// TwinCAT 3 PLC project Untitled1
// ProgramVersion: 3.1.4026.16
// libraries:
//   Tc2_MC2, * (Beckhoff Automation GmbH)
//   Tc2_Standard, * (Beckhoff Automation GmbH)
//   Tc2_System, * (Beckhoff Automation GmbH)
// project tree:
//   / PlcTask.TcTTO
//   POUs/ f_noteDecoder.TcPOU, MAIN.TcPOU, fb_MUZIK_Parser.TcPOU, nota_hiz_donusturucu.TcPOU, STRING_in_ARRAY.TcPOU
// real-time tasks:
//   TASK PlcTask: cycle T#10ms, priority 20, ADS port 350

CONFIGURATION Untitled1
    RESOURCE PLC ON TwinCAT3
        TASK PlcTask(INTERVAL := T#10ms, PRIORITY := 20);
        PROGRAM MAIN WITH PlcTask : MAIN;
    END_RESOURCE
END_CONFIGURATION

// ---- POUs/MAIN.TcPOU
PROGRAM MAIN
VAR
	b_butonlar 	: ARRAY[1..15] OF BOOL;
	r_zamanlar 	: ARRAY[1..15] OF REAL;
	b_togglelar : ARRAY[1..15] OF BOOL;
	b_scale		: ARRAY[1..12] OF BOOL;

	r_key		: REAL;

	i			: INT;
	j 			: INT := 1;
	k			: INT := 1;
	key_count	: INT;
	last_key	: INT;
	direction   : INT := 1;
	style		: INT;
	b_style		: BOOL;
	b_oldStyle  : BOOL;

	r_mm 		: REAL;
	r_offset	: REAL;
	r_Timer		: REAL;

	mcPower		:MC_Power;
	motor1		:AXIS_REF;
	mcJog		:MC_Jog;
	r_acceleration : REAL := 90000;
	r_deceleration : REAL := 40000;

	b_Manuel  	: BOOL;
	b_vibrato	: BOOL;
	b_Muzik		: BOOL;
	b_Otomatik	: BOOL;
	b_Major		: BOOL := TRUE;

	s_MajorMinor: STRING := 'Major';
	b_ScaleMajor: ARRAY[1..12] OF BOOL := [TRUE, FALSE, TRUE, FALSE, TRUE, TRUE, FALSE, TRUE, FALSE, TRUE, FALSE, TRUE];
	b_ScaleMinor: ARRAY[1..12] OF BOOL := [TRUE, FALSE, TRUE, TRUE, FALSE, TRUE, FALSE, TRUE, TRUE, FALSE, TRUE, FALSE];

	MUZIK_BPS 	: REAL := 10;
	OTOMATIK_BPS: REAL := 1;

	r_BPMTimer 	: REAL;
	r_timerOffset : REAL;
	r_noteTimer	: REAL;

	MUZIK_Parser : fb_MUZIK_Parser;

	MuzikCalmaTuru : BOOL := TRUE;

	(* Offset = -2 yap *)
	MUZIK		: ARRAY[1..100] OF REAL := [1, 1, 1, 5, 5, 5, 8, 8, 6, 6, 6, 10, 10, 10, 13, 13, 1, 1, 1, 5, 5, 5, 8, 8, 6, 13, 12, 13, 12, 13, 8, 5, 1, 1, 1, 5, 5, 5, 8, 8, 6, 6, 6, 10, 10, 10, 13, 13, 1, 1, 16, 16, 16, 15, 15, 15, 13, 13, 13, 8, 7, 8, 7, 4, -1];
	M_TETRIS 	: STRING(255)	 := ['A - E F G - F E D - D F A - G F E - - F G - A - F - D - D -*4 G - Bb D2 - C2 Bb A - - F A - G F E - E F G - A - F - D - D -*3'];
	M_CANAKKALE	: STRING(512) := ['E - Fs*2 -*2 Fs - Fs*10 E2*4 Eb2 E2 Eb2*3 E2*3 Db2*7 D2 Db2 B*3 Db2*6 Eb2*6 E2*6 Db2*6 B*19 -*5 B*3 Db2*3 -*3 Db2*2 - Db2*5 - Db2*3 B*2 - B*5 - B C2*2 B C2 B A*3 Ab*3 A*5 - Ab*3 A*3 B*3 A*3 C2*3 B*3 A*3 Ab*3 Fs*9 E*3 Ab*3 A*3 B*3 Db2*3 -*3 A*5 - Ab*2 - Ab*2 - Fs*8 - Fs*12 - Fs -*18'];
END_VAR

IF NOT (b_Muzik OR b_Otomatik) THEN
	r_mm := 0;
END_IF

(* Piyano tuşlarıyla çalma *)
IF b_Manuel THEN
	FOR i := 1 TO 15 DO
		IF b_butonlar[i] THEN
			r_zamanlar[i] := r_zamanlar[i] + 0.01;
	
			IF i = 1 THEN
				r_mm := nota_hiz_donusturucu(i, r_offset);
			ELSE
				IF (r_zamanlar[i] < r_zamanlar[i-1] AND r_zamanlar[i-1] > 0) OR r_zamanlar[i-1] = 0 THEN
					r_mm := nota_hiz_donusturucu(i, r_offset);
				END_IF
			END_IF
		ELSE
			r_zamanlar[i] := 0;
		END_IF
	END_FOR
END_IF



(* MUZIK'te kayıtlı müziği çalma  -----ESKI----- *)
IF b_Muzik AND NOT MuzikCalmaTuru THEN
	r_BPMTimer := r_BPMTimer + 0.01;
	IF r_BPMTimer > 1/MUZIK_BPS THEN
		r_BPMTimer := 0;
		j := j + 1;
	END_IF

	IF MUZIK[j] = -1 THEN
		j := 1;
	END_IF
	IF MUZIK[j] > 0 THEN
		r_MM := nota_hiz_donusturucu(MUZIK[j], r_offset);
	END_IF
END_IF



(* Daha iyi müzik çalar *)
IF b_Muzik AND MuzikCalmaTuru THEN
	r_offset := -2;
	IF r_noteTimer > 0 THEN
		r_noteTimer := r_noteTimer - 0.01;
	END_IF

	r_BPMTimer := r_BPMTimer + 0.01;
	IF r_BPMTimer > 1/MUZIK_BPS + SEL(r_mm = 0, 0, r_timerOffset) THEN
		r_BPMTimer := SEL(r_mm = 0, 0.0, r_timerOffset);
		MUZIK_Parser(
			MUZIK 		:= M_CANAKKALE,
			i_next 		:= TRUE,
			r_OFFSET	:= r_offset,
			b_stop 		:= FALSE,);
	END_IF
	IF MUZIK_Parser.newNote THEN
		r_noteTimer := 0.02;
	END_IF
	r_MM := MUZIK_Parser.r_mm + ((r_noteTimer) * -6000);
END_IF



(* Anahtar ve gam  *)
r_key := 0;
FOR i := 1 TO 12 DO
	IF b_scale[i] THEN
		r_key := i;
	END_IF
END_FOR

IF r_key > 0 THEN
	FOR i := 0 TO 11 DO
		key_count := REAL_TO_INT(r_key) + i;
		IF key_count > 12 THEN
			key_count := key_count - 12;
		END_IF
		IF b_Major THEN
			b_togglelar[key_count] := b_ScaleMajor[i+1];
		ELSE
			b_togglelar[key_count] := b_ScaleMinor[i+1];
		END_IF
	END_FOR
	b_togglelar[13] := b_togglelar[1];
	b_togglelar[14] := FALSE;
	b_togglelar[15] := FALSE;
END_IF


IF b_style AND NOT b_oldStyle THEN
	IF style > 1 THEN
		style := 0;
	ELSE
		style := style + 1;
	END_IF
END_IF
b_oldStyle := b_style;

(* Otomatik arpej *)
s_MajorMinor := SEL(b_Major, 'Minor', 'Major');
IF b_Otomatik THEN


	IF r_BPMTimer > 1/OTOMATIK_BPS THEN
		r_BPMTimer := 0;

		key_count := 0;
		REPEAT
			k := k + direction;
			IF k > 15 OR k < 1 THEN
				CASE style OF
					0 :
						k := 1;
						direction :=1;
					1 :
						k := 15;
						direction := -1;
					2 :
						direction := -direction;
						k := k + 2*direction;
				END_CASE
			END_IF
			key_count := key_count + 1;
		UNTIL  key_count > 20 OR (b_togglelar[k] AND last_key <> k)
		END_REPEAT
	END_IF
	IF b_togglelar[k] THEN
		last_key := k;
		r_mm := nota_hiz_donusturucu(k, r_offset);
	ELSE
		r_mm := 0;
	END_IF
	r_BPMTimer := r_BPMTimer + 0.01;
END_IF



(* Vibrato *)
IF b_vibrato AND r_mm > 0 THEN
	r_mm := LIMIT(0, r_mm + SIN(r_timer * 360*8 * (pi/180)) * 200, 8800);
END_IF
r_Timer := r_Timer + 0.01;




mcPower(
	Axis:= motor1,
	Enable:= TRUE,
	Enable_Positive:= TRUE,
	Enable_Negative:= TRUE,
	Override:= r_mm/9000 * 100,
	BufferMode:= MC_Aborting);

mcJog(
	Axis:= motor1,
	JogForward:= (r_mm > 0) AND mcPower.Status,
	JogBackwards:= FALSE,
	Mode:= MC_JOGMODE_CONTINOUS,
	Position:= 0,
	Velocity:= 9000,
	Acceleration:= r_acceleration,
	Deceleration:= r_deceleration,
	Jerk:= 900000);

END_PROGRAM

// ---- POUs/fb_MUZIK_Parser.TcPOU
FUNCTION_BLOCK fb_MUZIK_Parser
VAR_INPUT
	MUZIK 		: STRING(512);
	i_next 		: BOOL;
	r_OFFSET	: REAL;
	b_stop   	: BOOL := TRUE;
END_VAR
VAR_OUTPUT
	r_mm 		: REAL;
	newNote		: BOOL;
END_VAR
VAR
	char 		: STRING(4);
	s_reading	: STRING;
	s_NOTE		: STRING;
	r_OCTAVE	: REAL;
	s_OCTARR	: ARRAY[1..10] OF STRING(4) := ['0', '1', '2'];
	i			: INT;
	i_counter	: INT;
END_VAR

IF i_next THEN
	i_counter := i_counter - 1;

	IF i_counter < 1 THEN
		newNote := TRUE;
		s_reading := '';
		r_OCTAVE := 1;
		REPEAT
			i := i + 1;
			char := MID(MUZIK, 1, i);
			IF STRING_in_ARRAY(char, s_OCTARR) THEN
				r_OCTAVE := STRING_TO_REAL(char);
			ELSE
				s_reading := CONCAT(s_reading, char);
			END_IF
		UNTIL MID(MUZIK, 1, i+1) = ' ' OR MID(MUZIK, 1, i+1) = '*' OR i+1 > LEN(MUZIK)
		END_REPEAT

		i := i + 1;

		IF i >= LEN(MUZIK) THEN
			i := 0;
		END_IF

		s_NOTE := s_reading;

		IF MID(MUZIK, 1, i) = '*' THEN
			s_reading := '';
			REPEAT
				i := i + 1;
				char := MID(MUZIK, 1, i);
				s_reading := CONCAT(s_reading, char);
			UNTIL MID(MUZIK, 1, i+1) = ' ' OR i+1 > LEN(MUZIK)
			END_REPEAT
			i := i + 1;
			IF i >= LEN(MUZIK) THEN
				r_mm := 0;
				i:= 0;
			END_IF

			i_counter := STRING_TO_INT(s_reading);
		END_IF
	ELSE
		newNote := FALSE;
	END_IF

	IF s_NOTE = '-' OR s_NOTE = 'x' THEN
		newNote := FALSE;
		IF b_stop THEN
			r_mm := 0;
		END_IF
	ELSE
		r_mm := f_noteDecoder(s_NOTE, r_OCTAVE, r_OFFSET);
	END_IF
END_IF

END_FUNCTION_BLOCK

// ---- POUs/STRING_in_ARRAY.TcPOU
FUNCTION STRING_in_ARRAY : BOOL
VAR_INPUT
	s_STRING 	: STRING;
	s_ARRAY		: ARRAY[1..10] OF STRING(4);
END_VAR
VAR
	i 			: INT;
END_VAR

FOR i := 1 TO 10 DO
	IF s_ARRAY[i] = s_STRING THEN
		STRING_in_ARRAY := TRUE;
		RETURN;
		
	ELSIF s_ARRAY[i] = '' THEN
		STRING_in_ARRAY := FALSE;
		RETURN;
	END_IF
END_FOR

STRING_in_ARRAY := FALSE;
RETURN;

END_FUNCTION

// ---- POUs/f_noteDecoder.TcPOU
FUNCTION f_noteDecoder : REAL
VAR_INPUT
	s_NOTE 		: STRING;
	r_OCTAVE	: REAL;	
	r_OFFSET	: REAL;
END_VAR
VAR
	nota_01 : ARRAY[1..10] OF STRING(4)  := ['0', 'DO', 'C'];
	nota_02 : ARRAY[1..10] OF STRING(4)  := ['1', 'DO#', 'DOd', 'DOs', 'C#', 'Cd', 'Cs', 'REb', 'Db'];
	nota_03 : ARRAY[1..10] OF STRING(4)  := ['2', 'RE', 'D'];
	nota_04 : ARRAY[1..10] OF STRING(4)  := ['3', 'RE#', 'REd', 'REs', 'D#', 'Dd', 'Ds', 'MIb', 'Eb'];
	nota_05 : ARRAY[1..10] OF STRING(4)  := ['4', 'MI', 'E'];
	nota_06 : ARRAY[1..10] OF STRING(4)  := ['5', 'FA', 'F'];
	nota_07 : ARRAY[1..10] OF STRING(4)  := ['6', 'FA#', 'FAd', 'FAs', 'F#', 'Fd', 'Fs', 'SOLb', 'Gb'];
	nota_08 : ARRAY[1..10] OF STRING(4)  := ['7', 'SOL', 'G'];
	nota_09 : ARRAY[1..10] OF STRING(4)  := ['8', 'SOL#', 'SOLd', 'SOLs', 'G#', 'Gd', 'Gs', 'LAb', 'Ab'];
	nota_10 : ARRAY[1..10] OF STRING(4)  := ['9', 'LA', 'A'];
	nota_11 : ARRAY[1..10] OF STRING(4)  := ['10', 'LA#', 'LAd', 'LAs', 'A#', 'Ad', 'As', 'SIb', 'Bb'];
	nota_12 : ARRAY[1..10] OF STRING(4)  := ['11', 'SI', 'B'];
END_VAR

r_OCTAVE := r_OCTAVE - 1;
IF    STRING_in_ARRAY(s_NOTE, nota_01) THEN
	f_noteDecoder := nota_hiz_donusturucu(1  + (12 * r_OCTAVE), r_OFFSET);
ELSIF STRING_in_ARRAY(s_NOTE, nota_02) THEN
	f_noteDecoder := nota_hiz_donusturucu(2  + (12 * r_OCTAVE), r_OFFSET);
ELSIF STRING_in_ARRAY(s_NOTE, nota_03) THEN
	f_noteDecoder := nota_hiz_donusturucu(3  + (12 * r_OCTAVE), r_OFFSET);
ELSIF STRING_in_ARRAY(s_NOTE, nota_04) THEN
	f_noteDecoder := nota_hiz_donusturucu(4  + (12 * r_OCTAVE), r_OFFSET);
ELSIF STRING_in_ARRAY(s_NOTE, nota_05) THEN
	f_noteDecoder := nota_hiz_donusturucu(5  + (12 * r_OCTAVE), r_OFFSET);
ELSIF STRING_in_ARRAY(s_NOTE, nota_06) THEN
	f_noteDecoder := nota_hiz_donusturucu(6  + (12 * r_OCTAVE), r_OFFSET);
ELSIF STRING_in_ARRAY(s_NOTE, nota_07) THEN
	f_noteDecoder := nota_hiz_donusturucu(7  + (12 * r_OCTAVE), r_OFFSET);
ELSIF STRING_in_ARRAY(s_NOTE, nota_08) THEN
	f_noteDecoder := nota_hiz_donusturucu(8  + (12 * r_OCTAVE), r_OFFSET);
ELSIF STRING_in_ARRAY(s_NOTE, nota_09) THEN
	f_noteDecoder := nota_hiz_donusturucu(9  + (12 * r_OCTAVE), r_OFFSET);
ELSIF STRING_in_ARRAY(s_NOTE, nota_10) THEN
	f_noteDecoder := nota_hiz_donusturucu(10 + (12 * r_OCTAVE), r_OFFSET);
ELSIF STRING_in_ARRAY(s_NOTE, nota_11) THEN
	f_noteDecoder := nota_hiz_donusturucu(11 + (12 * r_OCTAVE), r_OFFSET);
ELSIF STRING_in_ARRAY(s_NOTE, nota_12) THEN
	f_noteDecoder := nota_hiz_donusturucu(12 + (12 * r_OCTAVE), r_OFFSET);
ELSE
	f_noteDecoder := 0;
END_IF

END_FUNCTION

// ---- POUs/nota_hiz_donusturucu.TcPOU
FUNCTION nota_hiz_donusturucu : REAL
VAR_INPUT
	nota :REAL;
	offset : REAL;
END_VAR

nota_hiz_donusturucu := LIMIT(0, (((((nota + offset)+8.845)*((nota + offset)+8.845)/9.708) + 29.03139) * 100), 8800);

END_FUNCTION
